% RSLogix 500 project WONDERFUL DRYER ORIGINAL_BAK006.RSS, saved by version 11.00.00.00 %
PROJECT "ML1400"    % processor: MicroLogix 1400; MAIN_PROG %

PROGRAM FILES
  LAD 2 "MAIN_PROG"  11 rungs
  LAD 3   10 rungs
  LAD 4   32 rungs
  LAD 5   8 rungs
  LAD 6   16 rungs
  LAD 7   2 rungs
  LAD 8   47 rungs
  LAD 9   2 rungs
  LAD 10   5 rungs
  LAD 11   17 rungs

DATA FILES
  O0 OUTPUT  10 elements
  I1 INPUT  23 elements
  S2 STATUS  66 elements
  B3 BINARY  20 elements
  T4 TIMER  11 elements
  C5 COUNTER  1 elements
  R6 CONTROL  1 elements
  N7 INTEGER  77 elements
  F8 FLOAT  1 elements
  PD9   2 elements

LADDER 2 "MAIN_PROG"
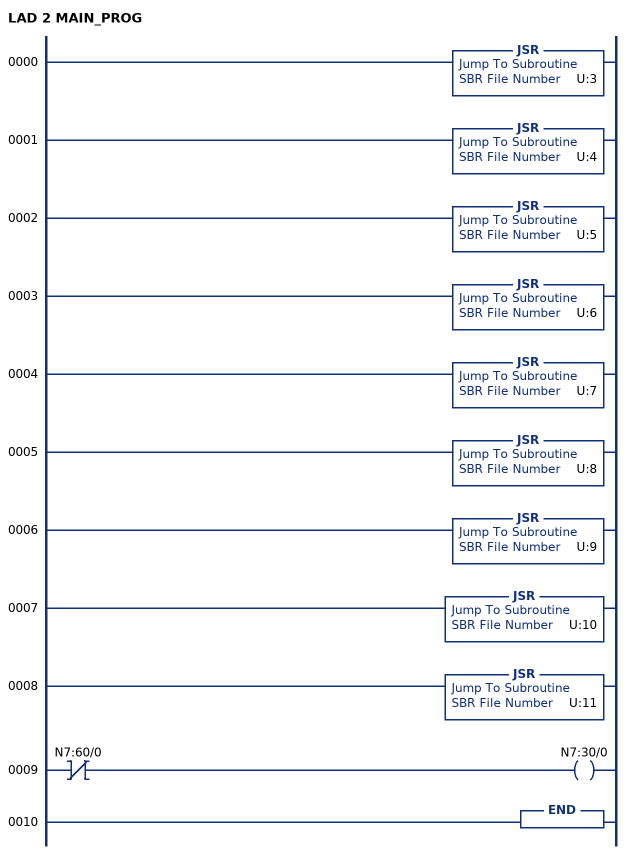
% Rung: 0 %
SOR JSR U:3 EOR
% Rung: 1 %
SOR JSR U:4 EOR
% Rung: 2 %
SOR JSR U:5 EOR
% Rung: 3 %
SOR JSR U:6 EOR
% Rung: 4 %
SOR JSR U:7 EOR
% Rung: 5 %
SOR JSR U:8 EOR
% Rung: 6 %
SOR JSR U:9 EOR
% Rung: 7 %
SOR JSR U:10 EOR
% Rung: 8 %
SOR JSR U:11 EOR
% Rung: 9 %
SOR XIO N7:60/0 OTE N7:30/0 EOR
% Rung: 10 %
SOR END EOR

LADDER 3
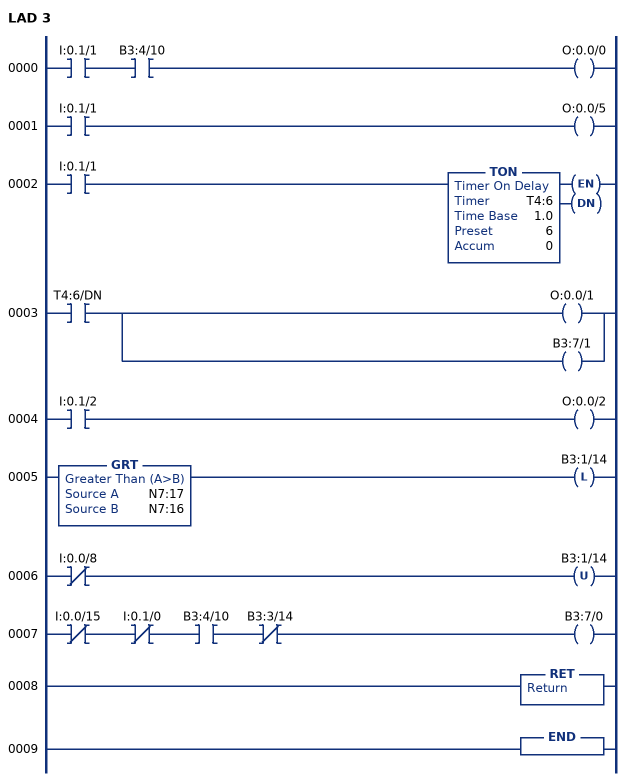
% Rung: 0 %
SOR XIC I:0.1/1 XIC B3:4/10 OTE O:0.0/0 EOR
% Rung: 1 %
SOR XIC I:0.1/1 OTE O:0.0/5 EOR
% Rung: 2 %
SOR XIC I:0.1/1 TON T4:6 1.0 6 0 EOR
% Rung: 3 %
SOR XIC T4:6/DN BST OTE O:0.0/1 NXB OTE B3:7/1 BND EOR
% Rung: 4 %
SOR XIC I:0.1/2 OTE O:0.0/2 EOR
% Rung: 5 %
SOR GRT N7:17 N7:16 OTL B3:1/14 EOR
% Rung: 6 %
SOR XIO I:0.0/8 OTU B3:1/14 EOR
% Rung: 7 %
SOR XIO I:0.0/15 XIO I:0.1/0 XIC B3:4/10 XIO B3:3/14 OTE B3:7/0 EOR
% Rung: 8 %
SOR RET EOR
% Rung: 9 %
SOR END EOR

LADDER 4
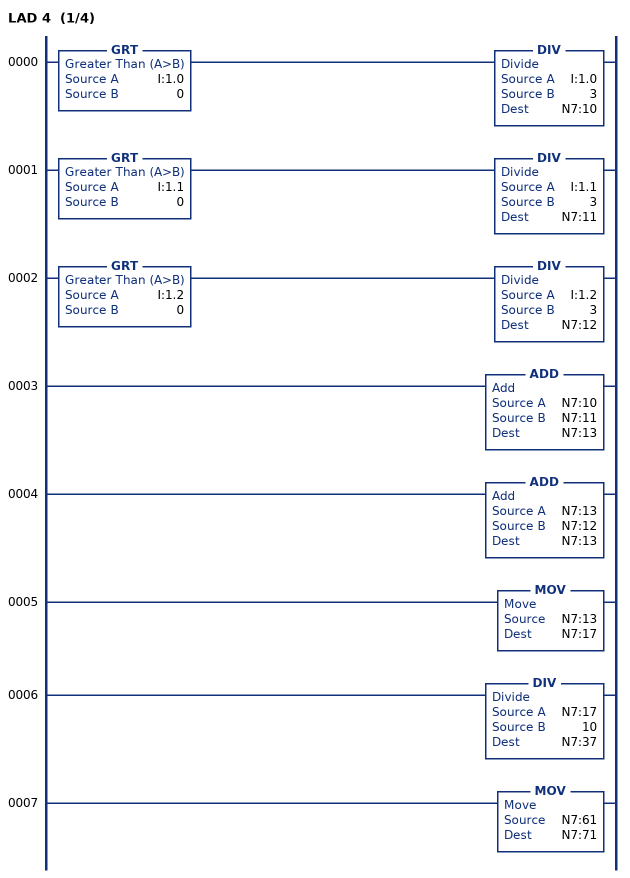
% Rung: 0 %
SOR GRT I:1.0 0 DIV I:1.0 3 N7:10 EOR
% Rung: 1 %
SOR GRT I:1.1 0 DIV I:1.1 3 N7:11 EOR
% Rung: 2 %
SOR GRT I:1.2 0 DIV I:1.2 3 N7:12 EOR
% Rung: 3 %
SOR ADD N7:10 N7:11 N7:13 EOR
% Rung: 4 %
SOR ADD N7:13 N7:12 N7:13 EOR
% Rung: 5 %
SOR MOV N7:13 N7:17 EOR
% Rung: 6 %
SOR DIV N7:17 10 N7:37 EOR
% Rung: 7 %
SOR MOV N7:61 N7:71 EOR

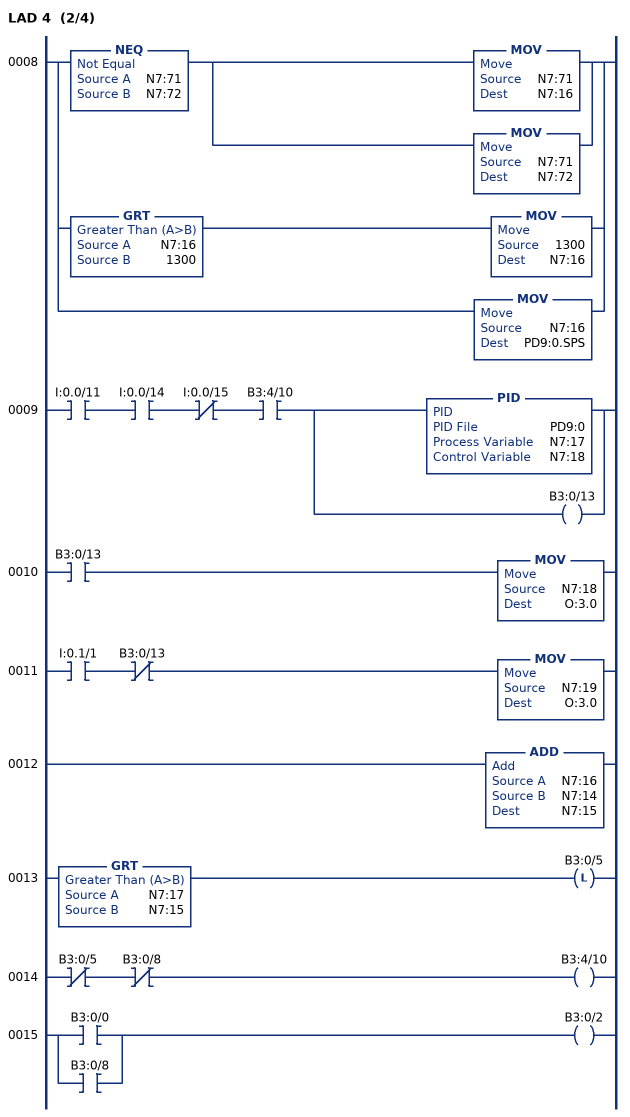
% Rung: 8 %
SOR BST NEQ N7:71 N7:72 BST MOV N7:71 N7:16 NXB MOV N7:71 N7:72 BND NXB GRT N7:16 1300 MOV 1300 N7:16 NXB MOV N7:16 PD9:0.SPS BND EOR
% Rung: 9 %
SOR XIC I:0.0/11 XIC I:0.0/14 XIO I:0.0/15 XIC B3:4/10 BST PID PD9:0 N7:17 N7:18 NXB OTE B3:0/13 BND EOR
% Rung: 10 %
SOR XIC B3:0/13 MOV N7:18 O:3.0 EOR
% Rung: 11 %
SOR XIC I:0.1/1 XIO B3:0/13 MOV N7:19 O:3.0 EOR
% Rung: 12 %
SOR ADD N7:16 N7:14 N7:15 EOR
% Rung: 13 %
SOR GRT N7:17 N7:15 OTL B3:0/5 EOR
% Rung: 14 %
SOR XIO B3:0/5 XIO B3:0/8 OTE B3:4/10 EOR
% Rung: 15 %
SOR BST XIC B3:0/0 NXB XIC B3:0/8 BND OTE B3:0/2 EOR

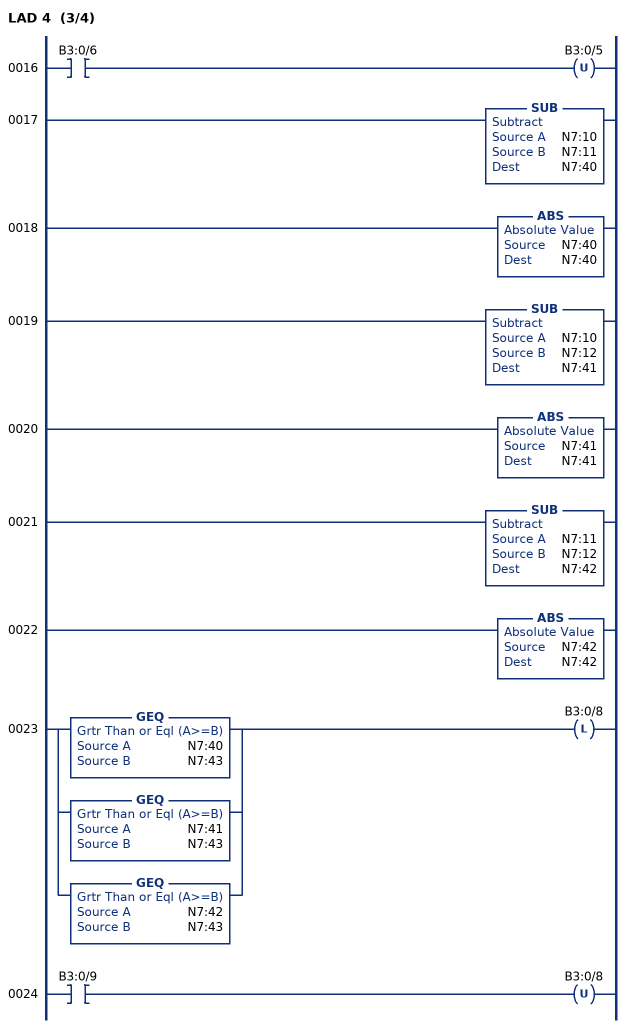
% Rung: 16 %
SOR XIC B3:0/6 OTU B3:0/5 EOR
% Rung: 17 %
SOR SUB N7:10 N7:11 N7:40 EOR
% Rung: 18 %
SOR ABS N7:40 N7:40 EOR
% Rung: 19 %
SOR SUB N7:10 N7:12 N7:41 EOR
% Rung: 20 %
SOR ABS N7:41 N7:41 EOR
% Rung: 21 %
SOR SUB N7:11 N7:12 N7:42 EOR
% Rung: 22 %
SOR ABS N7:42 N7:42 EOR
% Rung: 23 %
SOR BST GEQ N7:40 N7:43 NXB BST GEQ N7:41 N7:43 NXB GEQ N7:42 N7:43 BND BND OTL B3:0/8 EOR
% Rung: 24 %
SOR XIC B3:0/9 OTU B3:0/8 EOR

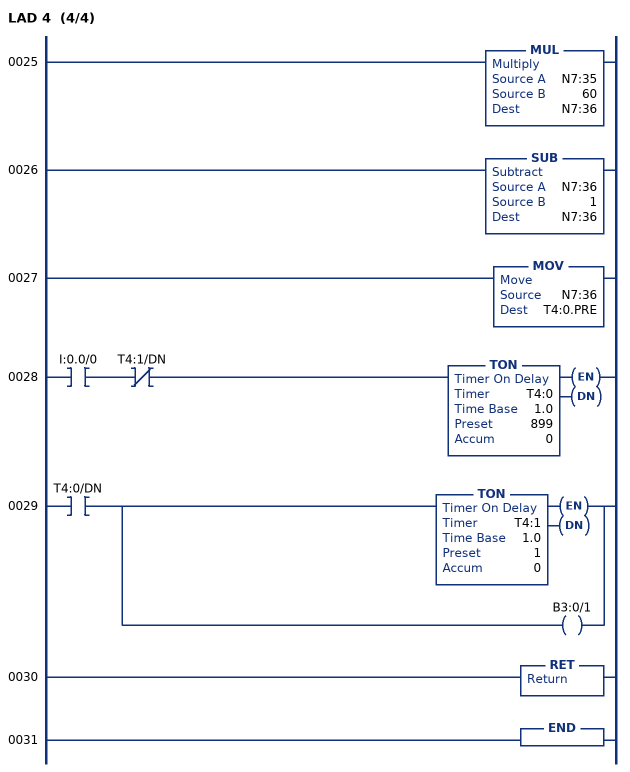
% Rung: 25 %
SOR MUL N7:35 60 N7:36 EOR
% Rung: 26 %
SOR SUB N7:36 1 N7:36 EOR
% Rung: 27 %
SOR MOV N7:36 T4:0.PRE EOR
% Rung: 28 %
SOR XIC I:0.0/0 XIO T4:1/DN TON T4:0 1.0 899 0 EOR
% Rung: 29 %
SOR XIC T4:0/DN BST TON T4:1 1.0 1 0 NXB OTE B3:0/1 BND EOR
% Rung: 30 %
SOR RET EOR
% Rung: 31 %
SOR END EOR

LADDER 5
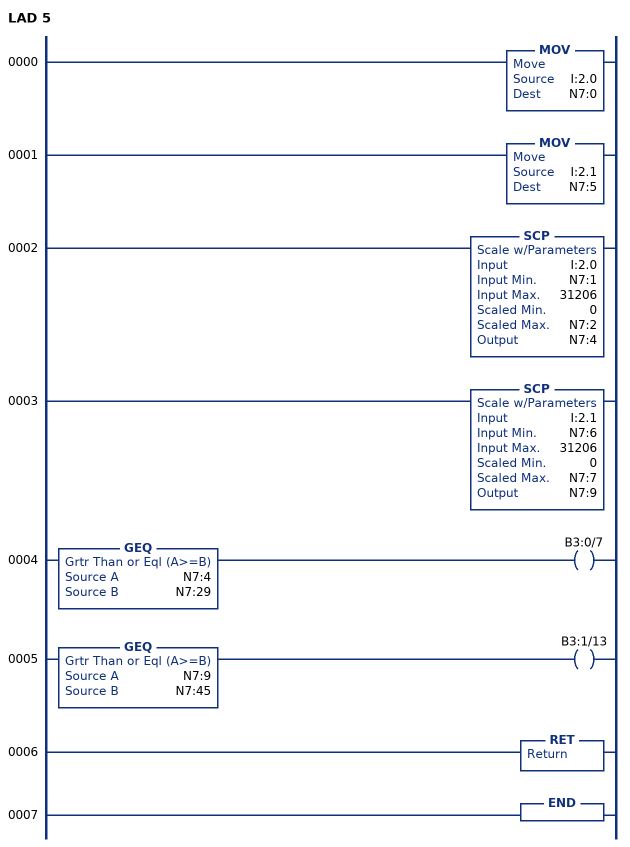
% Rung: 0 %
SOR MOV I:2.0 N7:0 EOR
% Rung: 1 %
SOR MOV I:2.1 N7:5 EOR
% Rung: 2 %
SOR SCP I:2.0 N7:1 31206 0 N7:2 N7:4 EOR
% Rung: 3 %
SOR SCP I:2.1 N7:6 31206 0 N7:7 N7:9 EOR
% Rung: 4 %
SOR GEQ N7:4 N7:29 OTE B3:0/7 EOR
% Rung: 5 %
SOR GEQ N7:9 N7:45 OTE B3:1/13 EOR
% Rung: 6 %
SOR RET EOR
% Rung: 7 %
SOR END EOR

LADDER 6
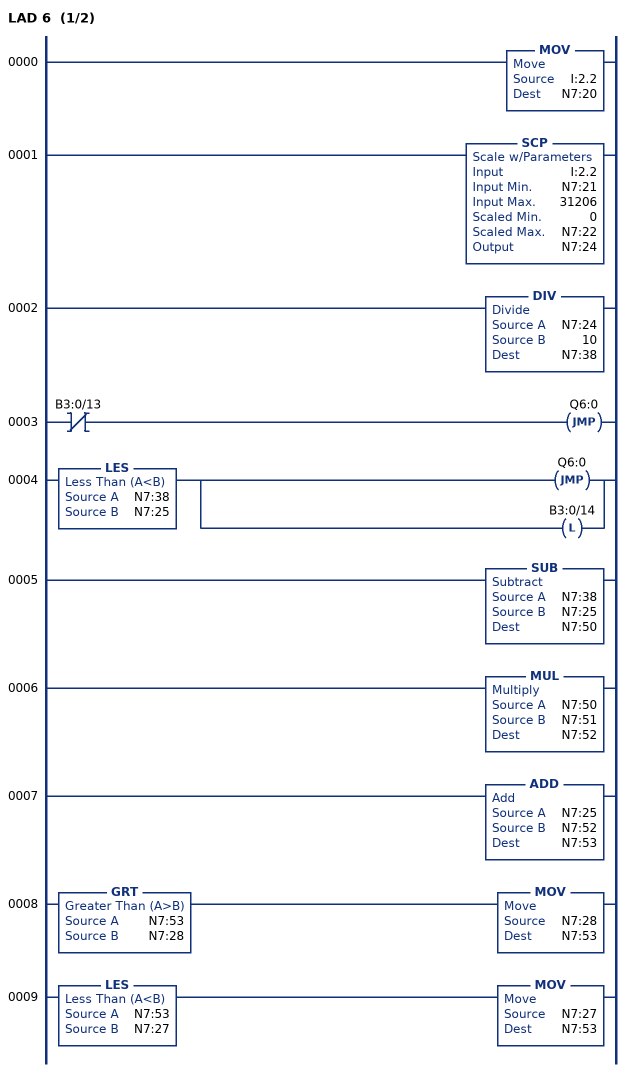
% Rung: 0 %
SOR MOV I:2.2 N7:20 EOR
% Rung: 1 %
SOR SCP I:2.2 N7:21 31206 0 N7:22 N7:24 EOR
% Rung: 2 %
SOR DIV N7:24 10 N7:38 EOR
% Rung: 3 %
SOR XIO B3:0/13 JMP Q6:0 EOR
% Rung: 4 %
SOR LES N7:38 N7:25 BST JMP Q6:0 NXB OTL B3:0/14 BND EOR
% Rung: 5 %
SOR SUB N7:38 N7:25 N7:50 EOR
% Rung: 6 %
SOR MUL N7:50 N7:51 N7:52 EOR
% Rung: 7 %
SOR ADD N7:25 N7:52 N7:53 EOR
% Rung: 8 %
SOR GRT N7:53 N7:28 MOV N7:28 N7:53 EOR
% Rung: 9 %
SOR LES N7:53 N7:27 MOV N7:27 N7:53 EOR

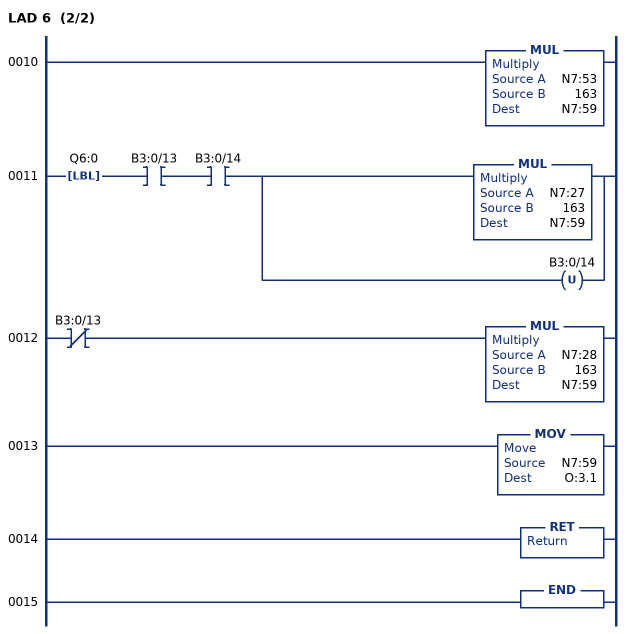
% Rung: 10 %
SOR MUL N7:53 163 N7:59 EOR
% Rung: 11 %
SOR LBL Q6:0 XIC B3:0/13 XIC B3:0/14 BST MUL N7:27 163 N7:59 NXB OTU B3:0/14 BND EOR
% Rung: 12 %
SOR XIO B3:0/13 MUL N7:28 163 N7:59 EOR
% Rung: 13 %
SOR MOV N7:59 O:3.1 EOR
% Rung: 14 %
SOR RET EOR
% Rung: 15 %
SOR END EOR

LADDER 7
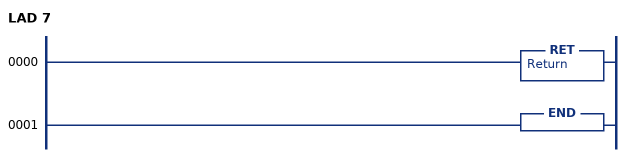
% Rung: 0 %
SOR RET EOR
% Rung: 1 %
SOR END EOR

LADDER 8
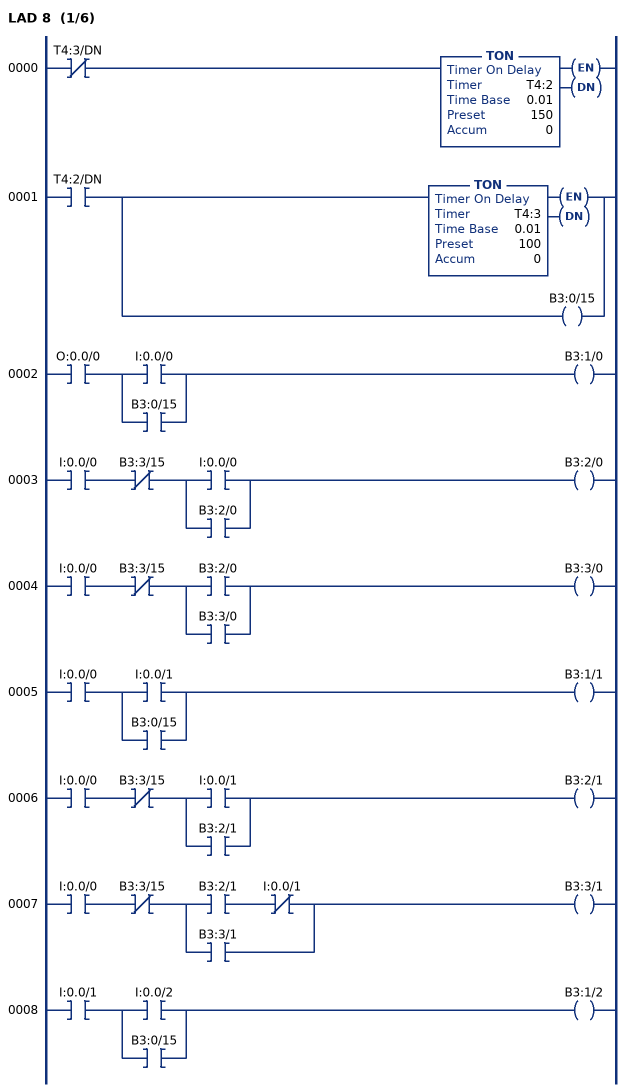
% Rung: 0 %
SOR XIO T4:3/DN TON T4:2 0.01 150 0 EOR
% Rung: 1 %
SOR XIC T4:2/DN BST TON T4:3 0.01 100 0 NXB OTE B3:0/15 BND EOR
% Rung: 2 %
SOR XIC O:0.0/0 BST XIC I:0.0/0 NXB XIC B3:0/15 BND OTE B3:1/0 EOR
% Rung: 3 %
SOR XIC I:0.0/0 XIO B3:3/15 BST XIC I:0.0/0 NXB XIC B3:2/0 BND OTE B3:2/0 EOR
% Rung: 4 %
SOR XIC I:0.0/0 XIO B3:3/15 BST XIC B3:2/0 NXB XIC B3:3/0 BND OTE B3:3/0 EOR
% Rung: 5 %
SOR XIC I:0.0/0 BST XIC I:0.0/1 NXB XIC B3:0/15 BND OTE B3:1/1 EOR
% Rung: 6 %
SOR XIC I:0.0/0 XIO B3:3/15 BST XIC I:0.0/1 NXB XIC B3:2/1 BND OTE B3:2/1 EOR
% Rung: 7 %
SOR XIC I:0.0/0 XIO B3:3/15 BST XIC B3:2/1 XIO I:0.0/1 NXB XIC B3:3/1 BND OTE B3:3/1 EOR
% Rung: 8 %
SOR XIC I:0.0/1 BST XIC I:0.0/2 NXB XIC B3:0/15 BND OTE B3:1/2 EOR

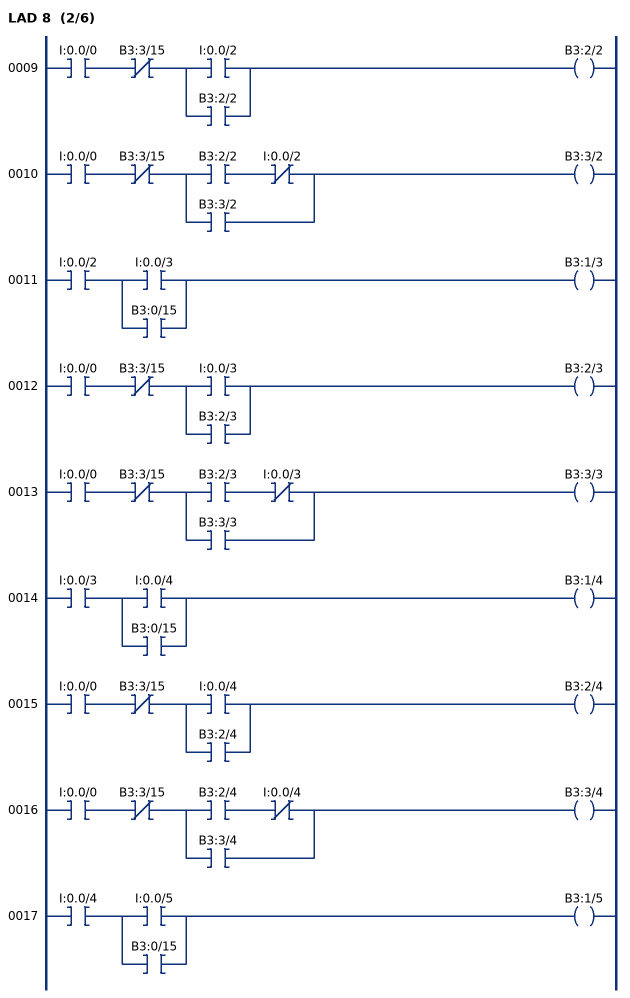
% Rung: 9 %
SOR XIC I:0.0/0 XIO B3:3/15 BST XIC I:0.0/2 NXB XIC B3:2/2 BND OTE B3:2/2 EOR
% Rung: 10 %
SOR XIC I:0.0/0 XIO B3:3/15 BST XIC B3:2/2 XIO I:0.0/2 NXB XIC B3:3/2 BND OTE B3:3/2 EOR
% Rung: 11 %
SOR XIC I:0.0/2 BST XIC I:0.0/3 NXB XIC B3:0/15 BND OTE B3:1/3 EOR
% Rung: 12 %
SOR XIC I:0.0/0 XIO B3:3/15 BST XIC I:0.0/3 NXB XIC B3:2/3 BND OTE B3:2/3 EOR
% Rung: 13 %
SOR XIC I:0.0/0 XIO B3:3/15 BST XIC B3:2/3 XIO I:0.0/3 NXB XIC B3:3/3 BND OTE B3:3/3 EOR
% Rung: 14 %
SOR XIC I:0.0/3 BST XIC I:0.0/4 NXB XIC B3:0/15 BND OTE B3:1/4 EOR
% Rung: 15 %
SOR XIC I:0.0/0 XIO B3:3/15 BST XIC I:0.0/4 NXB XIC B3:2/4 BND OTE B3:2/4 EOR
% Rung: 16 %
SOR XIC I:0.0/0 XIO B3:3/15 BST XIC B3:2/4 XIO I:0.0/4 NXB XIC B3:3/4 BND OTE B3:3/4 EOR
% Rung: 17 %
SOR XIC I:0.0/4 BST XIC I:0.0/5 NXB XIC B3:0/15 BND OTE B3:1/5 EOR

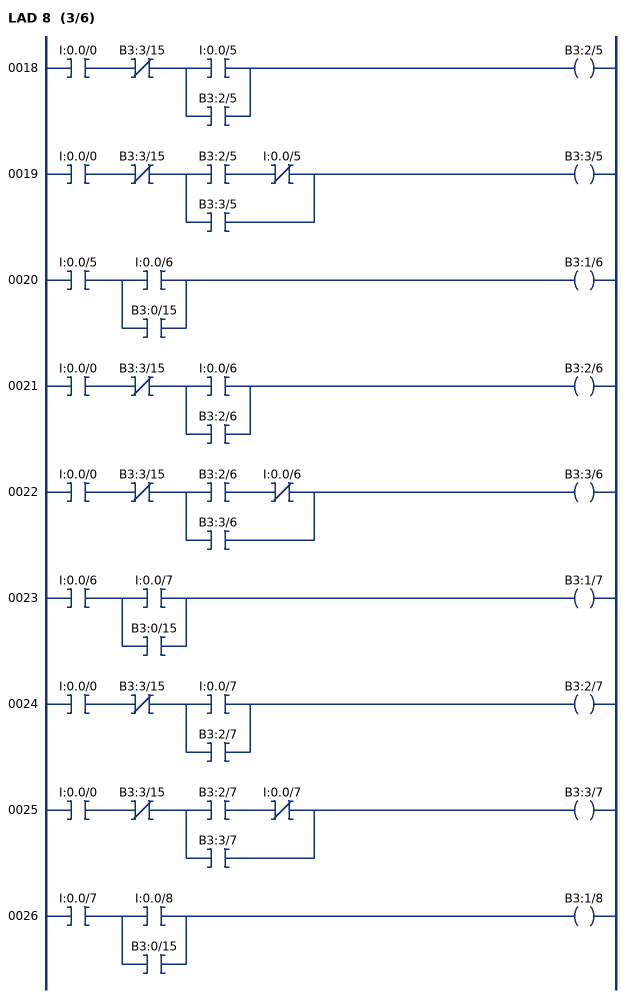
% Rung: 18 %
SOR XIC I:0.0/0 XIO B3:3/15 BST XIC I:0.0/5 NXB XIC B3:2/5 BND OTE B3:2/5 EOR
% Rung: 19 %
SOR XIC I:0.0/0 XIO B3:3/15 BST XIC B3:2/5 XIO I:0.0/5 NXB XIC B3:3/5 BND OTE B3:3/5 EOR
% Rung: 20 %
SOR XIC I:0.0/5 BST XIC I:0.0/6 NXB XIC B3:0/15 BND OTE B3:1/6 EOR
% Rung: 21 %
SOR XIC I:0.0/0 XIO B3:3/15 BST XIC I:0.0/6 NXB XIC B3:2/6 BND OTE B3:2/6 EOR
% Rung: 22 %
SOR XIC I:0.0/0 XIO B3:3/15 BST XIC B3:2/6 XIO I:0.0/6 NXB XIC B3:3/6 BND OTE B3:3/6 EOR
% Rung: 23 %
SOR XIC I:0.0/6 BST XIC I:0.0/7 NXB XIC B3:0/15 BND OTE B3:1/7 EOR
% Rung: 24 %
SOR XIC I:0.0/0 XIO B3:3/15 BST XIC I:0.0/7 NXB XIC B3:2/7 BND OTE B3:2/7 EOR
% Rung: 25 %
SOR XIC I:0.0/0 XIO B3:3/15 BST XIC B3:2/7 XIO I:0.0/7 NXB XIC B3:3/7 BND OTE B3:3/7 EOR
% Rung: 26 %
SOR XIC I:0.0/7 BST XIC I:0.0/8 NXB XIC B3:0/15 BND OTE B3:1/8 EOR

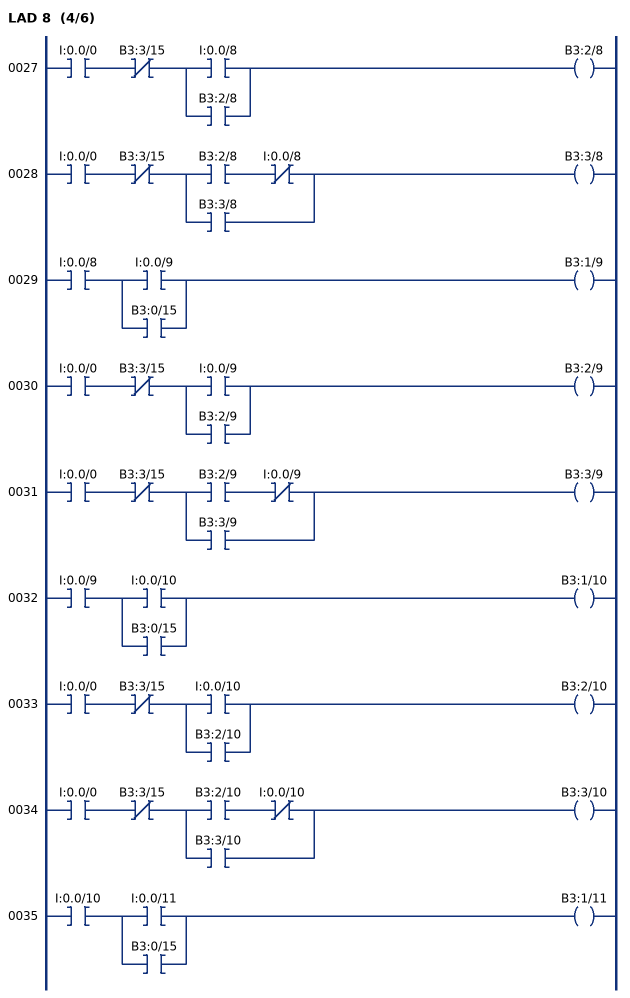
% Rung: 27 %
SOR XIC I:0.0/0 XIO B3:3/15 BST XIC I:0.0/8 NXB XIC B3:2/8 BND OTE B3:2/8 EOR
% Rung: 28 %
SOR XIC I:0.0/0 XIO B3:3/15 BST XIC B3:2/8 XIO I:0.0/8 NXB XIC B3:3/8 BND OTE B3:3/8 EOR
% Rung: 29 %
SOR XIC I:0.0/8 BST XIC I:0.0/9 NXB XIC B3:0/15 BND OTE B3:1/9 EOR
% Rung: 30 %
SOR XIC I:0.0/0 XIO B3:3/15 BST XIC I:0.0/9 NXB XIC B3:2/9 BND OTE B3:2/9 EOR
% Rung: 31 %
SOR XIC I:0.0/0 XIO B3:3/15 BST XIC B3:2/9 XIO I:0.0/9 NXB XIC B3:3/9 BND OTE B3:3/9 EOR
% Rung: 32 %
SOR XIC I:0.0/9 BST XIC I:0.0/10 NXB XIC B3:0/15 BND OTE B3:1/10 EOR
% Rung: 33 %
SOR XIC I:0.0/0 XIO B3:3/15 BST XIC I:0.0/10 NXB XIC B3:2/10 BND OTE B3:2/10 EOR
% Rung: 34 %
SOR XIC I:0.0/0 XIO B3:3/15 BST XIC B3:2/10 XIO I:0.0/10 NXB XIC B3:3/10 BND OTE B3:3/10 EOR
% Rung: 35 %
SOR XIC I:0.0/10 BST XIC I:0.0/11 NXB XIC B3:0/15 BND OTE B3:1/11 EOR

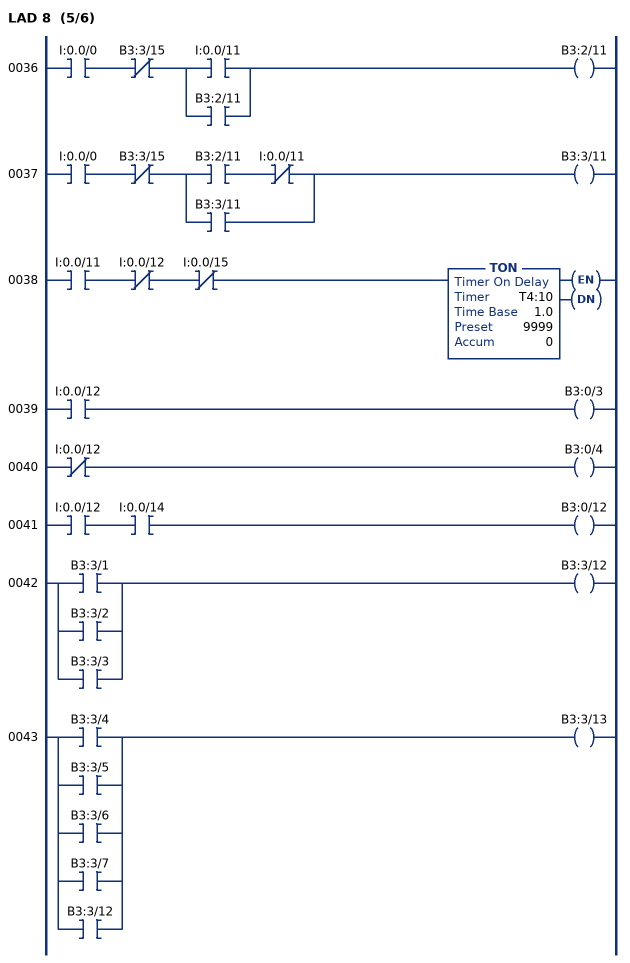
% Rung: 36 %
SOR XIC I:0.0/0 XIO B3:3/15 BST XIC I:0.0/11 NXB XIC B3:2/11 BND OTE B3:2/11 EOR
% Rung: 37 %
SOR XIC I:0.0/0 XIO B3:3/15 BST XIC B3:2/11 XIO I:0.0/11 NXB XIC B3:3/11 BND OTE B3:3/11 EOR
% Rung: 38 %
SOR XIC I:0.0/11 XIO I:0.0/12 XIO I:0.0/15 TON T4:10 1.0 9999 0 EOR
% Rung: 39 %
SOR XIC I:0.0/12 OTE B3:0/3 EOR
% Rung: 40 %
SOR XIO I:0.0/12 OTE B3:0/4 EOR
% Rung: 41 %
SOR XIC I:0.0/12 XIC I:0.0/14 OTE B3:0/12 EOR
% Rung: 42 %
SOR BST XIC B3:3/1 NXB BST XIC B3:3/2 NXB XIC B3:3/3 BND BND OTE B3:3/12 EOR
% Rung: 43 %
SOR BST XIC B3:3/4 NXB BST XIC B3:3/5 NXB BST XIC B3:3/6 NXB BST XIC B3:3/7 NXB XIC B3:3/12 BND BND BND BND OTE B3:3/13 EOR

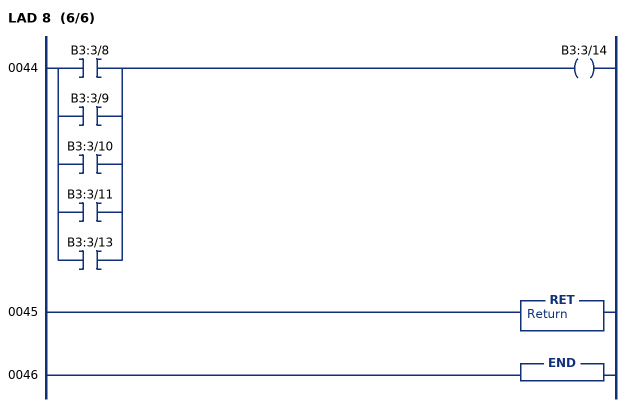
% Rung: 44 %
SOR BST XIC B3:3/8 NXB BST XIC B3:3/9 NXB BST XIC B3:3/10 NXB BST XIC B3:3/11 NXB XIC B3:3/13 BND BND BND BND OTE B3:3/14 EOR
% Rung: 45 %
SOR RET EOR
% Rung: 46 %
SOR END EOR

LADDER 9
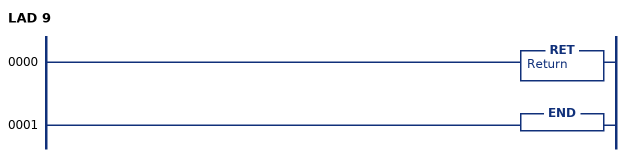
% Rung: 0 %
SOR RET EOR
% Rung: 1 %
SOR END EOR

LADDER 10
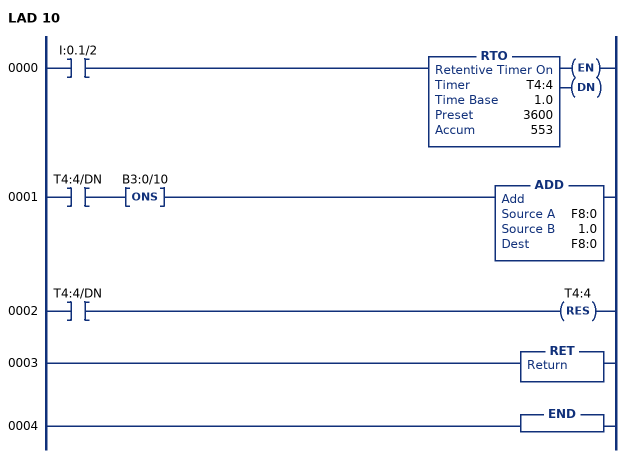
% Rung: 0 %
SOR XIC I:0.1/2 RTO T4:4 1.0 3600 553 EOR
% Rung: 1 %
SOR XIC T4:4/DN ONS B3:0/10 ADD F8:0 1.0 F8:0 EOR
% Rung: 2 %
SOR XIC T4:4/DN RES T4:4 EOR
% Rung: 3 %
SOR RET EOR
% Rung: 4 %
SOR END EOR

LADDER 11
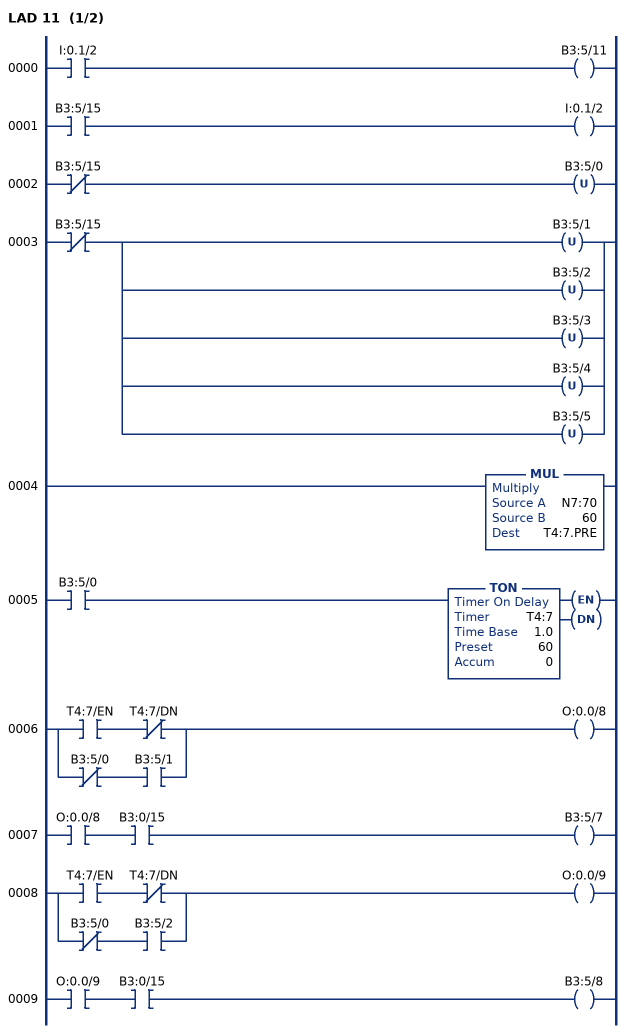
% Rung: 0 %
SOR XIC I:0.1/2 OTE B3:5/11 EOR
% Rung: 1 %
SOR XIC B3:5/15 OTE I:0.1/2 EOR
% Rung: 2 %
SOR XIO B3:5/15 OTU B3:5/0 EOR
% Rung: 3 %
SOR XIO B3:5/15 BST OTU B3:5/1 NXB BST OTU B3:5/2 NXB BST OTU B3:5/3 NXB BST OTU B3:5/4 NXB OTU B3:5/5 BND BND BND BND EOR
% Rung: 4 %
SOR MUL N7:70 60 T4:7.PRE EOR
% Rung: 5 %
SOR XIC B3:5/0 TON T4:7 1.0 60 0 EOR
% Rung: 6 %
SOR BST XIC T4:7/EN XIO T4:7/DN NXB XIO B3:5/0 XIC B3:5/1 BND OTE O:0.0/8 EOR
% Rung: 7 %
SOR XIC O:0.0/8 XIC B3:0/15 OTE B3:5/7 EOR
% Rung: 8 %
SOR BST XIC T4:7/EN XIO T4:7/DN NXB XIO B3:5/0 XIC B3:5/2 BND OTE O:0.0/9 EOR
% Rung: 9 %
SOR XIC O:0.0/9 XIC B3:0/15 OTE B3:5/8 EOR

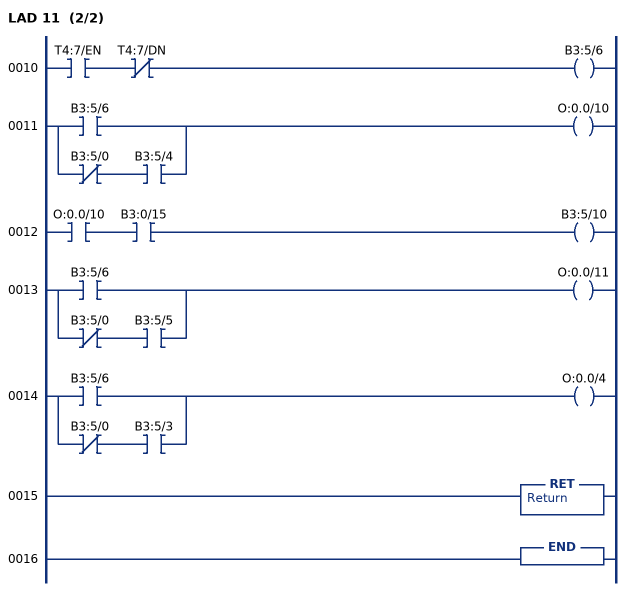
% Rung: 10 %
SOR XIC T4:7/EN XIO T4:7/DN OTE B3:5/6 EOR
% Rung: 11 %
SOR BST XIC B3:5/6 NXB XIO B3:5/0 XIC B3:5/4 BND OTE O:0.0/10 EOR
% Rung: 12 %
SOR XIC O:0.0/10 XIC B3:0/15 OTE B3:5/10 EOR
% Rung: 13 %
SOR BST XIC B3:5/6 NXB XIO B3:5/0 XIC B3:5/5 BND OTE O:0.0/11 EOR
% Rung: 14 %
SOR BST XIC B3:5/6 NXB XIO B3:5/0 XIC B3:5/3 BND OTE O:0.0/4 EOR
% Rung: 15 %
SOR RET EOR
% Rung: 16 %
SOR END EOR

REVISION NOTES
  0: Removed I:0/17 Normally closed

DATA TABLE (non-zero values as saved)
DATA B3
% B3:0 % 0X8010 0X8000 0X0000 0X0000 0X0580 0X0801 0X0000 0X0101 0X0000 0X0000
% B3:10 % 0X0001 0X0000 0X0000 0X0000 0X0000 0X0000 0X0000 0X0000 0X0000 0X0000
DATA T4
% .PRE .ACC %
% T4:0 % 899 0
% T4:1 % 1 0
% T4:2 % 150 0
% T4:3 % 100 0
% T4:4 % 3600 553
% T4:5 % 60 0
% T4:6 % 6 0
% T4:7 % 60 0
% T4:8 % 600 0
% T4:9 % 1800 0
% T4:10 % 9999 0
DATA N7
% N7:0 % 6194 6189 200 0 0 6177 6270 1188 0 -4
% N7:10 % 301 308 326 935 300 1500 1200 935 0 3277
% N7:20 % 6305 6250 1000 0 2 25 0 75 100 12
% N7:30 % 0 0 0 0 0 15 899 94 0 0
% N7:40 % 7 25 18 300 0 5 0 0 800 400
% N7:50 % 81 5 405 100 0 0 0 0 0 16300
% N7:60 % 1 1200 0 0 0 0 0 0 0 0
% N7:70 % 1 1200 1200 0 30 0 0
DATA F8
% F8:0 % 2580
